// TwinCAT 3 PLC project inovance_ctrl
// ProgramVersion: 3.1.4026.24
// libraries:
//   Tc2_MC2, * (Beckhoff Automation GmbH)
//   Tc2_Standard, * (Beckhoff Automation GmbH)
//   Tc2_System, * (Beckhoff Automation GmbH)
// project tree:
//   DUTs/ ST_AxisInternalSts.TcDUT, ST_HmiAxisCmd.TcDUT, ST_HmiAxisSet.TcDUT, ST_HmiAxisSts.TcDUT, ST_HmiComm.TcDUT
//   GVLs/ GVL_AxisCfg.TcGVL, GVL_AxisInternal.TcGVL, GVL_HMI.TcGVL
//   / PlcTask.TcTTO
//   POUs/ MAIN.TcPOU
// real-time tasks:
//   TASK PlcTask: cycle T#10ms, priority 20, ADS port 350
//   TASK PlcTask1: cycle T#10ms, priority 21, ADS port 351
// motion (NC):
//   TASK NC-Task 1 SAF: cycle T#2ms, priority 4, ADS port 501
//   TASK NC-Task 1 SVB: cycle T#10ms, priority 8, ADS port 511
//   AXIS 轴 1 (id 1)
//     OtherSettings: AllowMotionCmdToSlave=true
//     encoder EncType=19
//       EncPara: ScaleFactorNumerator=7.152557373e-06, MaxCount=#xffffffff
//     drive DrvType=16
//       DrvPara: MaxCount=#xffffffff, DriveControlDWord=#x00020100
//         Analog: TorqueSetpointScale=10, ScaleFactorActTorque=0.1
//         TimeComp: TaskDelayCycles=1
//     controller CtrType=1
//       CtrPara: PriorControlFactor=1
//         PosDiffControl: Range=20
//         Observer: BandWidth=20
// I/O:
//   DEVICE 设备 1 (EtherCAT), AmsNetId 172.18.238.251.2.1
//     驱动器 1 (InoSV660N) [SV660N_1Axis_00916]
// variable links:
//   NC-Task 1 SAF/Axes/轴 1 <-> 设备 1 (EtherCAT)/驱动器 1 (InoSV660N)
//     Drive/输入/In/nDataIn1 <-> Inputs/Following error actual value
//     Drive/输入/In/nDataIn3[0] <-> Inputs/Torque actual value
//     Drive/输入/In/nDcOutputTime <-> InfoData/DcOutputShift
//     Drive/输入/In/nState1 <-> Inputs/Statusword
//     Drive/输入/In/nState2 <-> Inputs/Statusword @bit 8
//     Drive/输入/In/nState4 @bit 1 <-> WcState/InputToggle
//     Drive/输入/In/nState4 <-> WcState/WcState
//     Drive/输出/Out/nCtrl1 <-> Outputs/Controlword
//     Drive/输出/Out/nCtrl2 <-> Outputs/Controlword @bit 8
//     Drive/输出/Out/nDataOut1 <-> Outputs/Target position
//     Enc/输入/In/nDataIn1 <-> Inputs/Position actual value
//     Enc/输入/In/nDataIn3 <-> Inputs/Touch probe pos1 pos value
//     Enc/输入/In/nDataIn5 <-> Inputs/Touch probe pos2 pos value
//     Enc/输入/In/nDcInputTime <-> InfoData/DcInputShift
//     Enc/输入/In/nState4 @bit 1 <-> WcState/InputToggle
//     Enc/输入/In/nState4 <-> WcState/WcState
//     Enc/输入/In/nState5 <-> Inputs/Touch probe status
//     Enc/输入/In/nState6 <-> Inputs/Touch probe status @bit 8
//     Enc/输出/Out/nCtrl5 <-> Outputs/Touch probe function
//     Enc/输出/Out/nCtrl6 <-> Outputs/Touch probe function @bit 8
//   inovance_ctrl/inovance_ctrl Instance <-> NC-Task 1 SAF/Axes/轴 1
//     PlcTask Inputs/MAIN.Axis_1.NcToPlc <-> 输出/ToPlc
//     PlcTask Outputs/MAIN.Axis_1.PlcToNc <-> 输入/FromPlc

CONFIGURATION inovance_ctrl
    RESOURCE PLC ON TwinCAT3
        TASK PlcTask(INTERVAL := T#10ms, PRIORITY := 21);
        PROGRAM MAIN WITH PlcTask : MAIN;
    END_RESOURCE
END_CONFIGURATION

// ---- DUTs/ST_AxisInternalSts.TcDUT
TYPE ST_AxisInternalSts :
STRUCT
    // Power 状态
    bPowerStatus       : BOOL;
    bPowerError        : BOOL;
    nPowerErrorID      : UDINT;

    // Reset 状态
    bResetBusy         : BOOL;
    bResetDone         : BOOL;
    bResetError        : BOOL;
    nResetErrorID      : UDINT;

    // 相对运动状态
    bMoveRelBusy       : BOOL;
    bMoveRelDone       : BOOL;
    bMoveRelError      : BOOL;
    nMoveRelErrorID    : UDINT;

    // 绝对运动状态
    bMoveAbsBusy       : BOOL;
    bMoveAbsDone       : BOOL;
    bMoveAbsError      : BOOL;
    nMoveAbsErrorID    : UDINT;

    // 点动速度运动状态
    bJogInVelocity     : BOOL;
    bJogBusy           : BOOL;
    bJogActive         : BOOL;
    bJogCommandAborted : BOOL;
    bJogError          : BOOL;
    nJogErrorID        : UDINT;

    // 点动 Halt 状态
    bJogHaltDone       : BOOL;
    bJogHaltBusy       : BOOL;
    bJogHaltActive     : BOOL;
    bJogHaltError      : BOOL;
    nJogHaltErrorID    : UDINT;

    // Stop 状态
    bStopDone          : BOOL;
    bStopBusy          : BOOL;
    bStopError         : BOOL;
    nStopErrorID       : UDINT;
END_STRUCT
END_TYPE

// ---- DUTs/ST_HmiAxisCmd.TcDUT
TYPE ST_HmiAxisCmd :
STRUCT
    bEnable  : BOOL;   // 伺服使能，保持型
    bReset   : BOOL;   // 轴复位，脉冲型，PLC 自动复位
    bStop    : BOOL;   // 软件停止，完成或报错后 PLC 自动复位

    bMoveRel : BOOL;   // 相对运动，脉冲型，PLC 自动复位
    bMoveAbs : BOOL;   // 绝对运动，脉冲型，PLC 自动复位

    bJogPos  : BOOL;   // 正向点动，HMI 按下 TRUE，松开 FALSE
    bJogNeg  : BOOL;   // 反向点动，HMI 按下 TRUE，松开 FALSE
END_STRUCT
END_TYPE

// ---- DUTs/ST_HmiAxisSet.TcDUT
TYPE ST_HmiAxisSet :
STRUCT
    fRelDistance : LREAL := 60.0;   // HMI 写入：相对运动距离
    fAbsPosition : LREAL := 0.0;    // HMI 写入：绝对运动目标位置
END_STRUCT
END_TYPE

// ---- DUTs/ST_HmiAxisSts.TcDUT
TYPE ST_HmiAxisSts :
STRUCT
    // 基本状态
    bPowerStatus : BOOL;     // 伺服是否使能
    bBusy        : BOOL;     // 轴总忙碌
    bError       : BOOL;     // 轴总报警
    nErrorID     : UDINT;    // 当前优先级最高的错误码

    // 运动状态编号
    // 0: Disabled/NotReady
    // 1: Standstill
    // 2: Moving
    // 3: Jogging
    // 4: Stopping
    // 5: Error
    // 6: Resetting
    nMotionState : INT;

    // 位置和速度
    fActPos      : LREAL;    // 实际位置
    fSetPos      : LREAL;    // 设定位置
    fActVelo     : LREAL;    // 实际速度，工程单位/s
    fActRpm      : LREAL;    // 实际转速，rpm
    fPosDiff     : LREAL;    // 设定位置 - 实际位置

    // 命令反馈，供 HMI 提示使用
    bCmdRejected : BOOL;     // 命令被拒绝，保持到下一次有效命令或复位
    nRejectReason: UDINT;    // 0 无；1 相对运动拒绝；2 绝对运动拒绝；3 正反点动冲突；4 点动条件不满足
END_STRUCT
END_TYPE

// ---- DUTs/ST_HmiComm.TcDUT
TYPE ST_HmiComm :
STRUCT
	udiHeartbeat : UDINT;   // HMI周期递增
    bOnline      : BOOL;    // PLC判断HMI是否在线
    bTimeout     : BOOL;    // PLC判断通信是否超时
END_STRUCT
END_TYPE

// ---- GVLs/GVL_AxisCfg.TcGVL
{attribute 'qualified_only'}
VAR_GLOBAL
    // 普通定位运动参数：由 PLC 底层控制，不开放给 HMI
    fMoveVelocity : LREAL := 60.0;
    fMoveAcc      : LREAL := 1000.0;
    fMoveDec      : LREAL := 1000.0;

    // 点动运动参数：由 PLC 底层控制，不开放给 HMI
    fJogVelocity  : LREAL := 60.0;
    fJogAcc       : LREAL := 500.0;
    fJogDec       : LREAL := 500.0;

    // 转速换算参数：若 60 mm = 1 rev，则 60 mm/s ≈ 60 rpm
    fMmPerRev     : LREAL := 60.0;

    // HMI 目标参数限幅
    fMaxRelDistance : LREAL := 6000.0;
    fMinRelDistance : LREAL := -6000.0;

    fMaxAbsPosition : LREAL := 6000.0;
    fMinAbsPosition : LREAL := -6000.0;
END_VAR

// ---- GVLs/GVL_AxisInternal.TcGVL
{attribute 'qualified_only'}
VAR_GLOBAL
    Axis1 : ST_AxisInternalSts;   // PLC 内部使用：功能块详细状态
END_VAR

// ---- GVLs/GVL_HMI.TcGVL
{attribute 'qualified_only'}
VAR_GLOBAL
    AxisCmd : ST_HmiAxisCmd;   // HMI/ADS 写入：命令
    AxisSet : ST_HmiAxisSet;   // HMI/ADS 写入：距离、位置
    AxisSts : ST_HmiAxisSts;   // HMI/ADS 读取：轴状态
	Comm : ST_HmiComm;		   //监控HMI通信状态
END_VAR

// ---- POUs/MAIN.TcPOU
PROGRAM MAIN
VAR
    Axis_1 : AXIS_REF;   // 在 TwinCAT 中与 NC 轴链接

    fbPower   : MC_Power;
    fbReset   : MC_Reset;
    fbMoveRel : MC_MoveRelative;
    fbMoveAbs : MC_MoveAbsolute;
    fbJogVel  : MC_MoveVelocity;
    fbJogHalt : MC_Halt;
    fbStop    : MC_Stop;

    trigReset      : R_TRIG;
    trigMoveRel    : R_TRIG;
    trigMoveAbs    : R_TRIG;
    trigJogRelease : F_TRIG;

    bBusyForNewCmd : BOOL;
    bBusyForJog    : BOOL;
    bErrorForCmd   : BOOL;

    bMoveRelExec   : BOOL;
    bMoveAbsExec   : BOOL;

    bJogExecute    : BOOL;
    bJogHaltReq    : BOOL;
    eJogDir        : MC_Direction := MC_Positive_Direction;

    fRelDistanceChecked : LREAL;
    fAbsPositionChecked : LREAL;
END_VAR

// =====================================================
// 1. 命令触发器
// =====================================================
trigReset(CLK := GVL_HMI.AxisCmd.bReset);
trigMoveRel(CLK := GVL_HMI.AxisCmd.bMoveRel);
trigMoveAbs(CLK := GVL_HMI.AxisCmd.bMoveAbs);

// =====================================================
// 2. HMI 目标参数限幅
// =====================================================
fRelDistanceChecked := GVL_HMI.AxisSet.fRelDistance;
IF fRelDistanceChecked > GVL_AxisCfg.fMaxRelDistance THEN
    fRelDistanceChecked := GVL_AxisCfg.fMaxRelDistance;
ELSIF fRelDistanceChecked < GVL_AxisCfg.fMinRelDistance THEN
    fRelDistanceChecked := GVL_AxisCfg.fMinRelDistance;
END_IF;

fAbsPositionChecked := GVL_HMI.AxisSet.fAbsPosition;
IF fAbsPositionChecked > GVL_AxisCfg.fMaxAbsPosition THEN
    fAbsPositionChecked := GVL_AxisCfg.fMaxAbsPosition;
ELSIF fAbsPositionChecked < GVL_AxisCfg.fMinAbsPosition THEN
    fAbsPositionChecked := GVL_AxisCfg.fMinAbsPosition;
END_IF;

// =====================================================
// 3. Reset 与 Power
// =====================================================
fbReset(
    Axis    := Axis_1,
    Execute := trigReset.Q,
    Done    => GVL_AxisInternal.Axis1.bResetDone,
    Busy    => GVL_AxisInternal.Axis1.bResetBusy,
    Error   => GVL_AxisInternal.Axis1.bResetError,
    ErrorID => GVL_AxisInternal.Axis1.nResetErrorID
);

IF trigReset.Q THEN
    GVL_HMI.AxisCmd.bReset := FALSE;
END_IF;

fbPower(
    Axis            := Axis_1,
    Enable          := GVL_HMI.AxisCmd.bEnable,
    Enable_Positive := TRUE,
    Enable_Negative := TRUE,
    Override        := 100.0,
    Status          => GVL_AxisInternal.Axis1.bPowerStatus,
    Error           => GVL_AxisInternal.Axis1.bPowerError,
    ErrorID         => GVL_AxisInternal.Axis1.nPowerErrorID
);

// =====================================================
// 4. 状态预处理：供本周期命令互锁使用
// =====================================================
bErrorForCmd := GVL_AxisInternal.Axis1.bPowerError
             OR GVL_AxisInternal.Axis1.bResetError
             OR GVL_AxisInternal.Axis1.bMoveRelError
             OR GVL_AxisInternal.Axis1.bMoveAbsError
             OR GVL_AxisInternal.Axis1.bStopError
             OR GVL_AxisInternal.Axis1.bJogError
             OR GVL_AxisInternal.Axis1.bJogHaltError;

bBusyForNewCmd := GVL_AxisInternal.Axis1.bResetBusy
               OR GVL_AxisInternal.Axis1.bMoveRelBusy
               OR GVL_AxisInternal.Axis1.bMoveAbsBusy
               OR GVL_AxisInternal.Axis1.bStopBusy
               OR GVL_AxisInternal.Axis1.bJogBusy
               OR GVL_AxisInternal.Axis1.bJogHaltBusy;

// 点动保持时不能被自身 bJogBusy 阻断，所以这里不包含 bJogBusy
bBusyForJog := GVL_AxisInternal.Axis1.bResetBusy
            OR GVL_AxisInternal.Axis1.bMoveRelBusy
            OR GVL_AxisInternal.Axis1.bMoveAbsBusy
            OR GVL_AxisInternal.Axis1.bStopBusy
            OR GVL_AxisInternal.Axis1.bJogHaltBusy;

// =====================================================
// 5. Stop 最高优先级：停止时取消点动命令和 Halt 请求
// =====================================================
IF GVL_HMI.AxisCmd.bStop THEN
    GVL_HMI.AxisCmd.bJogPos := FALSE;
    GVL_HMI.AxisCmd.bJogNeg := FALSE;
    bJogExecute := FALSE;
    bJogHaltReq := FALSE;
END_IF;

// =====================================================
// 6. 相对运动
// =====================================================
bMoveRelExec := trigMoveRel.Q
                AND NOT trigMoveAbs.Q
                AND GVL_AxisInternal.Axis1.bPowerStatus
                AND NOT bBusyForNewCmd
                AND NOT GVL_HMI.AxisCmd.bStop
                AND NOT GVL_HMI.AxisCmd.bJogPos
                AND NOT GVL_HMI.AxisCmd.bJogNeg
                AND NOT bErrorForCmd;

fbMoveRel(
    Axis         := Axis_1,
    Execute      := bMoveRelExec,
    Distance     := fRelDistanceChecked,
    Velocity     := GVL_AxisCfg.fMoveVelocity,
    Acceleration := GVL_AxisCfg.fMoveAcc,
    Deceleration := GVL_AxisCfg.fMoveDec,
    Done         => GVL_AxisInternal.Axis1.bMoveRelDone,
    Busy         => GVL_AxisInternal.Axis1.bMoveRelBusy,
    Error        => GVL_AxisInternal.Axis1.bMoveRelError,
    ErrorID      => GVL_AxisInternal.Axis1.nMoveRelErrorID
);

IF trigMoveRel.Q THEN
    GVL_HMI.AxisCmd.bMoveRel := FALSE;
END_IF;

// =====================================================
// 7. 绝对运动
// =====================================================
bMoveAbsExec := trigMoveAbs.Q
                AND NOT trigMoveRel.Q
                AND GVL_AxisInternal.Axis1.bPowerStatus
                AND NOT bBusyForNewCmd
                AND NOT GVL_HMI.AxisCmd.bStop
                AND NOT GVL_HMI.AxisCmd.bJogPos
                AND NOT GVL_HMI.AxisCmd.bJogNeg
                AND NOT bErrorForCmd;

fbMoveAbs(
    Axis         := Axis_1,
    Execute      := bMoveAbsExec,
    Position     := fAbsPositionChecked,
    Velocity     := GVL_AxisCfg.fMoveVelocity,
    Acceleration := GVL_AxisCfg.fMoveAcc,
    Deceleration := GVL_AxisCfg.fMoveDec,
    Done         => GVL_AxisInternal.Axis1.bMoveAbsDone,
    Busy         => GVL_AxisInternal.Axis1.bMoveAbsBusy,
    Error        => GVL_AxisInternal.Axis1.bMoveAbsError,
    ErrorID      => GVL_AxisInternal.Axis1.nMoveAbsErrorID
);

IF trigMoveAbs.Q THEN
    GVL_HMI.AxisCmd.bMoveAbs := FALSE;
END_IF;

// =====================================================
// 8. 点动 MoveVelocity
// =====================================================
bJogExecute := FALSE;

IF GVL_HMI.AxisCmd.bJogPos
   AND NOT GVL_HMI.AxisCmd.bJogNeg
   AND GVL_AxisInternal.Axis1.bPowerStatus
   AND NOT bBusyForJog
   AND NOT GVL_HMI.AxisCmd.bStop
   AND NOT bErrorForCmd THEN

    eJogDir := MC_Positive_Direction;
    bJogExecute := TRUE;

ELSIF GVL_HMI.AxisCmd.bJogNeg
      AND NOT GVL_HMI.AxisCmd.bJogPos
      AND GVL_AxisInternal.Axis1.bPowerStatus
      AND NOT bBusyForJog
      AND NOT GVL_HMI.AxisCmd.bStop
      AND NOT bErrorForCmd THEN

    eJogDir := MC_Negative_Direction;
    bJogExecute := TRUE;
ELSE
    bJogExecute := FALSE;
END_IF;

fbJogVel(
    Axis           := Axis_1,
    Execute        := bJogExecute,
    Velocity       := GVL_AxisCfg.fJogVelocity,
    Acceleration   := GVL_AxisCfg.fJogAcc,
    Deceleration   := GVL_AxisCfg.fJogDec,
    Direction      := eJogDir,
    InVelocity     => GVL_AxisInternal.Axis1.bJogInVelocity,
    Busy           => GVL_AxisInternal.Axis1.bJogBusy,
    Active         => GVL_AxisInternal.Axis1.bJogActive,
    CommandAborted => GVL_AxisInternal.Axis1.bJogCommandAborted,
    Error          => GVL_AxisInternal.Axis1.bJogError,
    ErrorID        => GVL_AxisInternal.Axis1.nJogErrorID
);

// =====================================================
// 9. 点动松手后 Halt
// =====================================================
trigJogRelease(CLK := bJogExecute);

IF trigJogRelease.Q AND NOT GVL_HMI.AxisCmd.bStop THEN
    bJogHaltReq := TRUE;
END_IF;

fbJogHalt(
    Axis         := Axis_1,
    Execute      := bJogHaltReq,
    Deceleration := GVL_AxisCfg.fJogDec,
    Done         => GVL_AxisInternal.Axis1.bJogHaltDone,
    Busy         => GVL_AxisInternal.Axis1.bJogHaltBusy,
    Active       => GVL_AxisInternal.Axis1.bJogHaltActive,
    Error        => GVL_AxisInternal.Axis1.bJogHaltError,
    ErrorID      => GVL_AxisInternal.Axis1.nJogHaltErrorID
);

IF GVL_AxisInternal.Axis1.bJogHaltDone OR GVL_AxisInternal.Axis1.bJogHaltError THEN
    bJogHaltReq := FALSE;
END_IF;

// =====================================================
// 10. Stop
// =====================================================
fbStop(
    Axis         := Axis_1,
    Execute      := GVL_HMI.AxisCmd.bStop,
    Deceleration := GVL_AxisCfg.fMoveDec,
    Done         => GVL_AxisInternal.Axis1.bStopDone,
    Busy         => GVL_AxisInternal.Axis1.bStopBusy,
    Error        => GVL_AxisInternal.Axis1.bStopError,
    ErrorID      => GVL_AxisInternal.Axis1.nStopErrorID
);

IF GVL_AxisInternal.Axis1.bStopDone OR GVL_AxisInternal.Axis1.bStopError THEN
    GVL_HMI.AxisCmd.bStop := FALSE;
END_IF;

// =====================================================
// 11. 命令拒绝提示
// =====================================================
IF trigReset.Q OR bMoveRelExec OR bMoveAbsExec OR GVL_HMI.AxisCmd.bStop OR bJogExecute THEN
    GVL_HMI.AxisSts.bCmdRejected := FALSE;
    GVL_HMI.AxisSts.nRejectReason := 0;
END_IF;

IF trigMoveRel.Q AND NOT bMoveRelExec THEN
    GVL_HMI.AxisSts.bCmdRejected := TRUE;
    GVL_HMI.AxisSts.nRejectReason := 1; // 相对运动命令被拒绝
ELSIF trigMoveAbs.Q AND NOT bMoveAbsExec THEN
    GVL_HMI.AxisSts.bCmdRejected := TRUE;
    GVL_HMI.AxisSts.nRejectReason := 2; // 绝对运动命令被拒绝
ELSIF GVL_HMI.AxisCmd.bJogPos AND GVL_HMI.AxisCmd.bJogNeg THEN
    GVL_HMI.AxisSts.bCmdRejected := TRUE;
    GVL_HMI.AxisSts.nRejectReason := 3; // 正反点动同时触发
    GVL_HMI.AxisCmd.bJogPos := FALSE;
    GVL_HMI.AxisCmd.bJogNeg := FALSE;
ELSIF (GVL_HMI.AxisCmd.bJogPos XOR GVL_HMI.AxisCmd.bJogNeg) AND NOT bJogExecute THEN
    GVL_HMI.AxisSts.bCmdRejected := TRUE;
    GVL_HMI.AxisSts.nRejectReason := 4; // 点动条件不满足
END_IF;

// =====================================================
// 12. HMI 状态汇总
// =====================================================
GVL_HMI.AxisSts.bPowerStatus := GVL_AxisInternal.Axis1.bPowerStatus;

GVL_HMI.AxisSts.fActPos  := Axis_1.NcToPlc.ActPos;
GVL_HMI.AxisSts.fSetPos  := Axis_1.NcToPlc.SetPos;
GVL_HMI.AxisSts.fActVelo := Axis_1.NcToPlc.ActVelo;

IF GVL_AxisCfg.fMmPerRev > 0.0 THEN
    GVL_HMI.AxisSts.fActRpm := GVL_HMI.AxisSts.fActVelo * 60.0 / GVL_AxisCfg.fMmPerRev;
ELSE
    GVL_HMI.AxisSts.fActRpm := 0.0;
END_IF;

GVL_HMI.AxisSts.fPosDiff := GVL_HMI.AxisSts.fSetPos - GVL_HMI.AxisSts.fActPos;

GVL_HMI.AxisSts.bBusy := GVL_AxisInternal.Axis1.bResetBusy
                      OR GVL_AxisInternal.Axis1.bMoveRelBusy
                      OR GVL_AxisInternal.Axis1.bMoveAbsBusy
                      OR GVL_AxisInternal.Axis1.bStopBusy
                      OR GVL_AxisInternal.Axis1.bJogBusy
                      OR GVL_AxisInternal.Axis1.bJogHaltBusy;

GVL_HMI.AxisSts.bError := GVL_AxisInternal.Axis1.bPowerError
                       OR GVL_AxisInternal.Axis1.bResetError
                       OR GVL_AxisInternal.Axis1.bMoveRelError
                       OR GVL_AxisInternal.Axis1.bMoveAbsError
                       OR GVL_AxisInternal.Axis1.bStopError
                       OR GVL_AxisInternal.Axis1.bJogError
                       OR GVL_AxisInternal.Axis1.bJogHaltError;

IF GVL_AxisInternal.Axis1.bPowerError THEN
    GVL_HMI.AxisSts.nErrorID := GVL_AxisInternal.Axis1.nPowerErrorID;
ELSIF GVL_AxisInternal.Axis1.bResetError THEN
    GVL_HMI.AxisSts.nErrorID := GVL_AxisInternal.Axis1.nResetErrorID;
ELSIF GVL_AxisInternal.Axis1.bMoveRelError THEN
    GVL_HMI.AxisSts.nErrorID := GVL_AxisInternal.Axis1.nMoveRelErrorID;
ELSIF GVL_AxisInternal.Axis1.bMoveAbsError THEN
    GVL_HMI.AxisSts.nErrorID := GVL_AxisInternal.Axis1.nMoveAbsErrorID;
ELSIF GVL_AxisInternal.Axis1.bStopError THEN
    GVL_HMI.AxisSts.nErrorID := GVL_AxisInternal.Axis1.nStopErrorID;
ELSIF GVL_AxisInternal.Axis1.bJogError THEN
    GVL_HMI.AxisSts.nErrorID := GVL_AxisInternal.Axis1.nJogErrorID;
ELSIF GVL_AxisInternal.Axis1.bJogHaltError THEN
    GVL_HMI.AxisSts.nErrorID := GVL_AxisInternal.Axis1.nJogHaltErrorID;
ELSE
    GVL_HMI.AxisSts.nErrorID := 0;
END_IF;

// 运动状态编号：0 Disabled, 1 Standstill, 2 Moving, 3 Jogging, 4 Stopping, 5 Error, 6 Resetting
IF GVL_HMI.AxisSts.bError THEN
    GVL_HMI.AxisSts.nMotionState := 5;
ELSIF NOT GVL_HMI.AxisSts.bPowerStatus THEN
    GVL_HMI.AxisSts.nMotionState := 0;
ELSIF GVL_AxisInternal.Axis1.bResetBusy THEN
    GVL_HMI.AxisSts.nMotionState := 6;
ELSIF GVL_AxisInternal.Axis1.bStopBusy OR GVL_AxisInternal.Axis1.bJogHaltBusy THEN
    GVL_HMI.AxisSts.nMotionState := 4;
ELSIF GVL_AxisInternal.Axis1.bJogBusy THEN
    GVL_HMI.AxisSts.nMotionState := 3;
ELSIF GVL_AxisInternal.Axis1.bMoveRelBusy OR GVL_AxisInternal.Axis1.bMoveAbsBusy THEN
    GVL_HMI.AxisSts.nMotionState := 2;
ELSE
    GVL_HMI.AxisSts.nMotionState := 1;
END_IF;

END_PROGRAM
